PROGRAM ReactorTemperature
VAR
	TemperatureControlStateMachine : FB_ReactorTemperatureControlStateMachine;
	_pidControllerParameters : ST_PidParameters;
	_manualControlPercentage : INT;
	_upperTemperature : INT;
	_lowerTemperature : INT;
	_temperatureSetpoint : INT;
	_temperatureContactor : BOOL;
	_autoControlSelected : BOOL;
	_temperatureContactorCommand : BOOL;
END_VAR


_upperTemperature	:= GVL_IO.reactorTemperatureUpper/10;
_lowerTemperature := GVL_IO.reactorTemperatureLower/10;
GVL_IO.reactorTemperatureContactor := _temperatureContactor;

// Temperature PID control logic
TemperatureControlStateMachine(temperatureMeasurement := TO_REAL(_upperTemperature),
							temperatureSetpoint := TO_REAL(_temperatureSetpoint),
							pidParameters := _pidControllerParameters,
							manualControlPercentage := _manualControlPercentage,
							autoControlSelected := _autoControlSelected,
							relayOn => _temperatureContactor);

IF _autoControlSelected OR (NOT _autoControlSelected AND _manualControlPercentage > 0) THEN
	_temperatureContactor := TemperatureControlStateMachine.relayOn;
ELSE
	_temperatureContactor := _temperatureContactorCommand;
END_IF

PROPERTY autoControlSelected : BOOL
SET

_autoControlSelected := autoControlSelected;
END_SET
END_PROPERTY

PROPERTY lowerTemperature : INT
GET

lowerTemperature := _lowerTemperature;
END_GET
END_PROPERTY

PROPERTY manualControlPercentage : INT
SET


_manualControlPercentage := manualControlPercentage;
END_SET
END_PROPERTY

PROPERTY pidControllerParameters : ST_PidParameters
SET

_pidControllerParameters := pidControllerParameters;
END_SET
END_PROPERTY

PROPERTY temperatureContactor : BOOL
GET

temperatureContactor := _temperatureContactor;
END_GET
END_PROPERTY

PROPERTY temperatureContactorCommand : BOOL
SET

_temperatureContactorCommand := temperatureContactorCommand;
END_SET
END_PROPERTY

PROPERTY temperatureSetpoint : INT
SET

_temperatureSetpoint := temperatureSetpoint;
END_SET
END_PROPERTY

PROPERTY upperTemperature : INT
GET

upperTemperature := _upperTemperature;
END_GET
END_PROPERTY

END_PROGRAM

(* stored: Version 1.1.0.1, ProductVersion 3.1.4024.9
   POU ReactorTemperature: Id {b264a75d-055d-45ef-ac02-67880535c654}, SpecialFunc None
   Property autoControlSelected: Id {7f26212f-80c2-4e14-963e-4ce92499c181}
   Set Set: Id {dc712bed-2067-4279-b7a8-706ce7b7d03d}
   Property lowerTemperature: Id {88abff98-3ec2-4bdc-9d32-aee098608a79}
   Get Get: Id {881f5bc1-ee7c-49fe-bce9-a74f34989737}
   Property manualControlPercentage: Id {ead5434f-49a2-4a32-8c04-ec55ff3a1e8a}
   Set Set: Id {c8e9bf7a-7b88-44b7-b4a9-b87d8a70468c}
   Property pidControllerParameters: Id {646e59c0-265d-4aea-9693-ebdf1d70de6c}
   Set Set: Id {74401392-871c-4c3a-b2a5-0ee58b8bde1d}
   Property temperatureContactor: Id {651aaa74-c7af-4155-91ce-d9b147209b1c}
   Get Get: Id {ed04c757-d4b1-4b51-bd63-6684d528cc07}
   Property temperatureContactorCommand: Id {be0d3024-09ac-474a-b153-44c6a5b42491}
   Set Set: Id {b728023f-4905-41fd-8922-03426fb04baf}
   Property temperatureSetpoint: Id {8e9d1647-23ef-4949-b863-ea810656227c}
   Set Set: Id {7c1326ac-99f1-4791-91f9-3ed3ce46bb17}
   Property upperTemperature: Id {84243da1-7d07-4d5a-b916-9af3257e9f21}
   Get Get: Id {56cb51bc-a137-41ac-aeee-448c455129d3} *)
